(* CoDeSys 2.3 export: BINSUBSTATUS.EXP *)

(* Data type in ENUM *)
TYPE BinSubStatus : (BinSubStatusNormal:=0, BinSubStatusSensorStopped, BinSubStatusRefStopped, BinSubStatusOverflow, BinSubStatusConfErr);
END_TYPE
